Universal Robots PolyScope program: test.urp

Program test (installation=string_planes directory=/programs createdIn=5.17.3 lastSavedIn=5.17.3 robotSerialNumber=20245501435)
Calibrated DH parameters: a=[0.000154, -0.137004, -0.385524, -0.00002, 0.000092, 0]; d=[0.162441, 211.794786, -230.585024, 18.923638, 0.099786, 0.09951]; alpha=[1.569493, -0.001902, 0.003874, 1.570111, -1.570167, 0]; deltaTheta=[0, -1.242934, 1.056292, 0.186646, 0.000002, 0.000001]
InitVariablesNode
Robot Program (runOnlyOnce=true)
  Call d_eighth
  Call d_eighthUp
SubProgram -> d_eighth
SubProgram -> d_eighthUp
SubProgram d_eighth (keepSynchronizedWithDisk=false) programFile=/programs/d_eighth.urp
  MoveL speed 250 mm/s, acceleration 1200 mm/s^2 (useActiveTCP=true) feature=Plane_2
    Waypoint Waypoint_5: TCP in base x=331.961 y=722.321 z=108.294 mm, rx=-1.6449 ry=-2.1081 rz=1.059 rad; joints [-129.708, -21.469, 51.981, -76.269, -76.861, -148.976] deg; TCP offset x=28.21 y=-96.107 z=-99.69 mm, rx=0 ry=0 rz=0 rad; feature pose in base x=343.605 y=747.803 z=100.778 mm, rx=2.7685 ry=0.1285 rz=1.3673 rad
    Waypoint Waypoint_1: TCP in base x=338.919 y=665.001 z=114.26 mm, rx=-1.6378 ry=-2.1148 rz=1.0804 rad; joints [-132.848, -27.946, 64.83, -81.449, -79.739, -151.46] deg
SubProgram d_eighthUp (keepSynchronizedWithDisk=false) programFile=/programs/d_eighthUp.urp
  MoveL speed 250 mm/s, acceleration 1200 mm/s^2 (useActiveTCP=true) feature=Plane_2
    Waypoint Waypoint_4: TCP in base x=338.919 y=665.001 z=114.26 mm, rx=-1.6378 ry=-2.1148 rz=1.0804 rad; joints [-132.848, -27.946, 64.83, -81.449, -79.739, -151.46] deg
    Waypoint Waypoint_2: TCP in base x=331.961 y=722.321 z=108.294 mm, rx=-1.6449 ry=-2.1081 rz=1.059 rad; joints [-129.708, -21.469, 51.981, -76.269, -76.861, -148.976] deg
